FUNCTION_BLOCK ButtonNC
VAR
	input AT %I* : BOOL;
END_VAR

PROPERTY IsPressed : BOOL
GET
IsPressed := input;
END_GET
END_PROPERTY

PROPERTY IsReleased : BOOL
GET
IsReleased := NOT input;
END_GET
END_PROPERTY

END_FUNCTION_BLOCK

(* stored: Version 1.1.0.1, ProductVersion 3.1.4024.12
   POU ButtonNC: Id {593d0c36-a778-4d44-b389-505244cedeb5}, SpecialFunc None
   Property IsPressed: Id {9d839024-b65a-4ac9-af8e-8dd66e30aabb}
   Get Get: Id {c882a1d8-fd95-4f7c-9833-b6b07ceec2d0}
   Property IsReleased: Id {0b008a41-96ec-4b7e-84e4-d431771c7175}
   Get Get: Id {adcd4b1c-2ed5-4aa7-9f23-40d8650a980a} *)
